INTERFACE I_MarkDefinition

(*
  Get a mark definition.
  nIdx= 1.._nMarks = registered marks
  nIdx= 0 - selects last mark 
  nIdx=-1 - selects boarder mark
*)
METHOD getMark : POINTER TO ST_MarkDefinition
VAR_INPUT
  nIdx : DINT; // mark index: 1.._nMarks, 0 = last (endMark) 
END_VAR
END_METHOD

(*Number of registered marks*)
PROPERTY nMarks : UDINT
GET
END_GET
END_PROPERTY

(*Number of detected marks*)
PROPERTY nMarksDetected : UDINT
GET
END_GET
END_PROPERTY

(*
  Register a mark to camera (teach)
*)
METHOD RegisterMark : BOOL
VAR_INPUT
  sMark : ST_MarkDefinition;
END_VAR
END_METHOD

METHOD ResetDefinition
END_METHOD

(*
  Reset all registered marks
*)
METHOD ResetMarkStates
END_METHOD

END_INTERFACE

(* stored: Version 1.1.0.1, ProductVersion 3.1.4024.11
   Itf I_MarkDefinition: Id {961e3342-2c28-4702-a1e0-dacac6afe5f8}
   Method getMark: Id {6dcce5ab-646c-4060-81c3-0eea54c1a7d3}
   Property nMarks: Id {f474363f-e035-45ba-8c0d-d254c1952798}
   Get Get: Id {de13454a-17e8-4b5c-b134-a5f1999f8846}
   Property nMarksDetected: Id {885555d1-3ee1-4fa8-9437-dc3e560f4a49}
   Get Get: Id {a6f0de8a-1ba3-4716-b602-4d6e217d2773}
   Method RegisterMark: Id {9eb8c8e0-d3b0-445a-b94d-730dc7ec70d1}
   Method ResetDefinition: Id {cdd0ec98-aac9-46a3-a823-70f18b7e54e9}
   Method ResetMarkStates: Id {8f025160-d4e0-46ad-879f-d784c19efaeb} *)
